PROGRAM PRG_LVCP5
VAR
END_VAR

	PRG_LVCP5_PowerMeasurement();

 	PRG_LVCP5_CompensationCalculate();

	PRG_LVCP5_MainCircuitBreaker();
	
	PRG_LVCP5_Colors();
	
	PRG_LVCP5_Group1();
	
	PRG_LVCP5_Group2();
	
	PRG_LVCP5_Group3();	
	
	PRG_LVCP5_Group4();	

	PRG_LVCP5_Group5();	

	PRG_LVCP5_Group6();	

	PRG_LVCP5_Group7();

END_PROGRAM

(* stored: Version 1.1.0.1, ProductVersion 3.1.4024.13
   POU PRG_LVCP5: Id {18ab8ba3-8ac4-4e40-a325-116379e8dbfa}, SpecialFunc None *)
